// TIA Portal V20 export
TYPE "LER_typeAlignThetaCalibrationConfiguration"
// stored: Access Published
   STRUCT
      MoveDeg : DInt;
      XPosition : Array[0..18] of LReal;
      Y1Position : Array[0..18] of LReal;
      Y2Position : Array[0..18] of LReal;
   END_STRUCT;
END_TYPE
